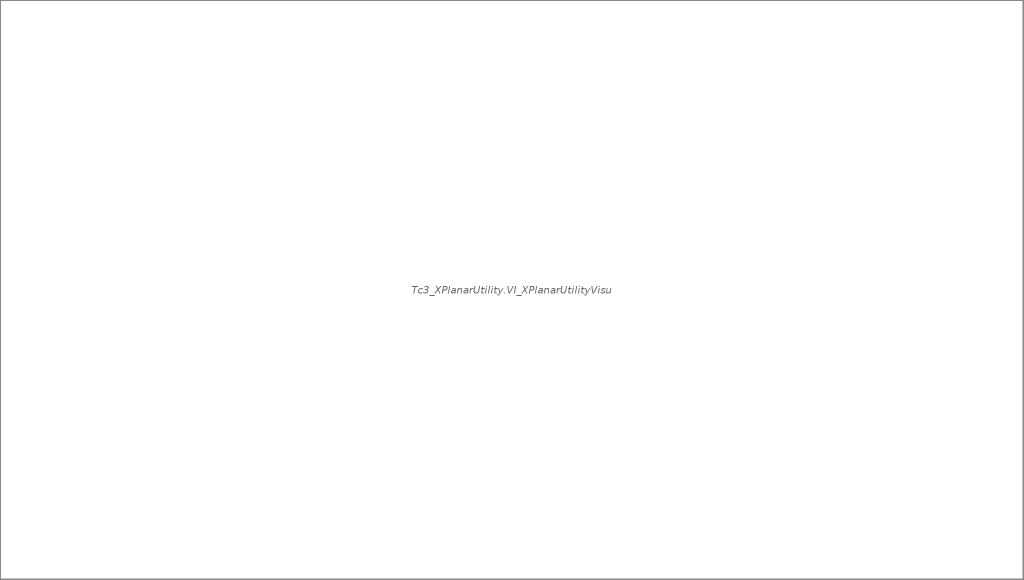
VISUALIZATION VI_Tc3_XPlanarUtility  // 1024x580
    Frame (0,0 1024x580)
        shows Tc3_XPlanarUtility.VI_XPlanarUtilityVisu()
END_VISUALIZATION

(* stored: Version 1.1.0.1, ProductVersion 3.1.4024.9
   Visu VI_Tc3_XPlanarUtility: Id {533de65a-912d-4635-99ac-138319ff7e7f} *)
